(* PLC project ia_tools test project, CODESYS CODESYS V3.5 SP16, author Toni Kucic *)
(* stored: creationDateTime 2021-03-31T21:46:16.9462712, version 1.0, modificationDateTime 2021-03-31T21:46:13.3815902, organization ia_tools *)
(* This is a test project to test and display the ia_tools features *)

TYPE typeDUT1 : STRUCT
  dummy1 : BOOL := TRUE;  (* Dummy variable1 *)
  dummy2 : REAL;  (* Dummy variable2 *)
  dummy3 : typeDUT2;  (* Dummy variable3 *)
  dummy4 : ARRAY[0..2] OF BOOL;  (* Dummy variable4 *)
END_STRUCT;
END_TYPE

TYPE typeDUT2 : STRUCT
  dummy1 : BOOL := TRUE;  (* Dummy variable1 *)
  dummy2 : REAL;  (* Dummy variable2 *)
  dummy3 : typeDUT1;  (* Dummy variable3 *)
  dummy4 : ARRAY[0..2] OF BOOL;  (* Dummy variable4 *)
END_STRUCT;
END_TYPE

(* values of enumTest: member1: Documentation of member 1; member2: Documentation of member 2; member3: Documentation of member 3; member4: Documentation of member 4 without value *)

{attribute 'qualified_only'}
{attribute 'strict'}
TYPE enumTest : (member1 := 0, member2 := 1, member3 := 3, member4);
END_TYPE

TYPE dummyDUT1 : STRUCT
  dummy1 : BOOL := TRUE;  (* Dummy variable1 *)
  dummy2 : REAL;  (* Dummy variable2 *)
  dummy3 : dummyDUT2;  (* Dummy variable3 *)
  dummy4 : ARRAY[0..2] OF BOOL;  (* Dummy variable4 *)
END_STRUCT;
END_TYPE

TYPE dummyDUT2 : STRUCT
  dummy1 : BOOL := TRUE;  (* Dummy variable1 *)
  dummy2 : REAL;  (* Dummy variable2 *)
  dummy3 : dummyDUT1;  (* Dummy variable3 *)
  dummy4 : ARRAY[0..2] OF BOOL;  (* Dummy variable4 *)
END_STRUCT;
END_TYPE

TYPE dummyDUT1 : STRUCT
  dummy1 : BOOL := TRUE;  (* Dummy variable1 *)
  dummy2 : REAL;  (* Dummy variable2 *)
  dummy3 : dummyDUT2;  (* Dummy variable3 *)
  dummy4 : ARRAY[0..2] OF BOOL;  (* Dummy variable4 *)
END_STRUCT;
END_TYPE

TYPE dummyDUT2 : STRUCT
  dummy1 : BOOL := TRUE;  (* Dummy variable1 *)
  dummy2 : REAL;  (* Dummy variable2 *)
  dummy3 : dummyDUT1;  (* Dummy variable3 *)
  dummy4 : ARRAY[0..2] OF BOOL;  (* Dummy variable4 *)
END_STRUCT;
END_TYPE

TYPE DUT : STRUCT

END_STRUCT;
END_TYPE

TYPE dummyDUT1 : STRUCT
  dummy1 : BOOL := TRUE;  (* Dummy variable1 *)
  dummy2 : REAL;  (* Dummy variable2 *)
  dummy3 : dummyDUT2;  (* Dummy variable3 *)
  dummy4 : ARRAY[0..2] OF BOOL;  (* Dummy variable4 *)
END_STRUCT;
END_TYPE

TYPE dummyDUT2 : STRUCT
  dummy1 : BOOL := TRUE;  (* Dummy variable1 *)
  dummy2 : REAL;  (* Dummy variable2 *)
  dummy3 : dummyDUT1;  (* Dummy variable3 *)
  dummy4 : ARRAY[0..2] OF BOOL;  (* Dummy variable4 *)
END_STRUCT;
END_TYPE

TYPE dummyDUT1 : STRUCT
  dummy1 : BOOL := TRUE;  (* Dummy variable1 *)
  dummy2 : REAL;  (* Dummy variable2 *)
  dummy3 : dummyDUT2;  (* Dummy variable3 *)
  dummy4 : ARRAY[0..2] OF BOOL;  (* Dummy variable4 *)
END_STRUCT;
END_TYPE

TYPE dummyDUT2 : STRUCT
  dummy1 : BOOL := TRUE;  (* Dummy variable1 *)
  dummy2 : REAL;  (* Dummy variable2 *)
  dummy3 : dummyDUT1;  (* Dummy variable3 *)
  dummy4 : ARRAY[0..2] OF BOOL;  (* Dummy variable4 *)
END_STRUCT;
END_TYPE

{attribute 'qualified_only'}
VAR_GLOBAL  (* typeGlobalList1 *)
  dummy1 : BOOL := TRUE;  (* Dummy variable1 *)
  dummy2 : REAL;  (* Dummy variable2 *)
  dummy3 : typeDUT1;  (* Dummy variable3 *)
  dummy4 : typeDUT2;  (* Dummy variable4 *)
  dummy5 : ARRAY[0..2] OF BOOL;  (* Dummy variable5 *)
  dummy6 : ARRAY[0..2] OF BOOL := [TRUE, FALSE, TRUE];  (* 1D array with initialization *)
  dummy7 : ARRAY[0..2, 0..3] OF INT;  (* 2D array without initialization *)
  dummy8 : ARRAY[0..2, 0..3] OF INT := [0, 1, 2, 3, 4, 5, 6, 7, 8];  (* 2D array with initialization *)
END_VAR

{attribute 'qualified_only'}
VAR_GLOBAL  (* typeGlobalList2 *)
  dummy1 : BOOL := TRUE;  (* Dummy variable1 *)
  dummy2 : REAL;  (* Dummy variable2 *)
  dummy3 : typeDUT1;  (* Dummy variable3 *)
  dummy4 : typeDUT2;  (* Dummy variable4 *)
  dummy5 : ARRAY[0..2] OF BOOL;  (* Dummy variable5 *)
END_VAR

PROGRAM typeProgram
  VAR_INPUT
    inputVar1 : BOOL;  (* Comment of inputVar1 *)
    inputVar2 : BOOL;  (* Comment of inputVar2 *)
    inputVar3 : POINTER TO BOOL;  (* Comment of inputVar3 as a pointer *)
  END_VAR
  VAR_IN_OUT
    inoutVar1 : BOOL;  (* Comment of inoutVar1 *)
    inoutVar2 : BOOL;  (* Comment of inoutVar2 *)
    inoutVar3 : POINTER TO BOOL;  (* Comment of inoutVar3 as a pointer *)
  END_VAR
  VAR_OUTPUT
    outputVar1 : BOOL;  (* Comment of outputVar1 *)
    outputVar2 : BOOL;  (* Comment of outputVar2 *)
    outputVar3 : POINTER TO BOOL;  (* Comment of outputVar3 as a pointer *)
  END_VAR
  VAR
    localVar1 : BOOL;  (* Comment of localVar1 *)
    localVar2 : BOOL;  (* Comment of localVar2 *)
    localVar3 : POINTER TO BOOL;  (* Local var as a pointer *)
  END_VAR

            (* THIS IS HOW THE CODE LOOKS *)

(*** DOCS STRING EXAMPLE ONE LINE***)
(*** DOCS STRING EXAMPLE
	MULTI
			LINE
			***)
(*** DOCS STRING WITH EMBEDDED CODE *)
outputVar1 := outputVar2;
(* THE CODE ABOVE IS INCLUDED IN THE DOCS ***)

          
END_PROGRAM

FUNCTION_BLOCK typeFunctionBlock
  VAR_INPUT
    inputVar1 : BOOL;  (* Comment of inputVar1 *)
    inputVar2 : BOOL;  (* Comment of inputVar2 *)
    inputVar3 : POINTER TO BOOL;  (* Comment of inputVar3 as a pointer *)
  END_VAR
  VAR_IN_OUT
    inoutVar1 : BOOL;  (* Comment of inoutVar1 *)
    inoutVar2 : BOOL;  (* Comment of inoutVar2 *)
    inoutVar3 : POINTER TO BOOL;  (* Comment of inoutVar3 as a pointer *)
  END_VAR
  VAR_OUTPUT
    outputVar1 : BOOL;  (* Comment of outputVar1 *)
    outputVar2 : BOOL;  (* Comment of outputVar2 *)
    outputVar3 : POINTER TO BOOL;  (* Comment of outputVar3 as a pointer *)
  END_VAR
  VAR
    localVar1 : BOOL;  (* Comment of localVar1 *)
    localVar2 : BOOL;  (* Comment of localVar2 *)
    localVar3 : POINTER TO BOOL;  (* Local var as a pointer *)
  END_VAR

            (* THIS IS HOW THE CODE LOOKS *)

(*** DOCS STRING EXAMPLE ONE LINE***)
(*** DOCS STRING EXAMPLE
	MULTI
			LINE
			***)
(*** DOCS STRING WITH EMBEDDED CODE *)
outputVar1 := outputVar2;
(* THE CODE ABOVE IS INCLUDED IN THE DOCS ***)

          
END_FUNCTION_BLOCK

FUNCTION typeFunction : BOOL
  VAR_INPUT
    inputVar1 : BOOL;  (* Comment of inputVar1 *)
    inputVar2 : BOOL;  (* Comment of inputVar2 *)
    inputVar3 : POINTER TO BOOL;  (* Comment of inputVar3 as a pointer *)
  END_VAR
  VAR_IN_OUT
    inoutVar1 : BOOL;  (* Comment of inoutVar1 *)
    inoutVar2 : BOOL;  (* Comment of inoutVar2 *)
    inoutVar3 : POINTER TO BOOL;  (* Comment of inoutVar3 as a pointer *)
  END_VAR
  VAR_OUTPUT
    outputVar1 : BOOL;  (* Comment of outputVar1 *)
    outputVar2 : BOOL;  (* Comment of outputVar2 *)
    outputVar3 : POINTER TO BOOL;  (* Comment of outputVar3 as a pointer *)
  END_VAR
  VAR
    localVar1 : BOOL;  (* Comment of localVar1 *)
    localVar2 : BOOL;  (* Comment of localVar2 *)
    localVar3 : POINTER TO BOOL;  (* Local var as a pointer to elementary value *)
    localVar4 : POINTER TO enumTest;  (* Local var as a pointer to enumeration *)
    localVar5 : POINTER TO typeDUT1;  (* Local var as a pointer to structure *)
    localVar6 : POINTER TO ARRAY[0..2] OF INT;  (* Local var as a pointer to structure *)
    localVar7 : typeDUT1 := (dummy1 := TRUE, dummy2 := 14.5);  (* Local var, structure with complex init *)
    dummy5 : ARRAY[0..2] OF BOOL;  (* Dummy variable5 *)
    dummy6 : ARRAY[0..2] OF BOOL := [TRUE, FALSE, TRUE];  (* 1D array with initialization *)
    dummy7 : ARRAY[0..2, 0..3] OF INT;  (* 2D array without initialization *)
    dummy8 : ARRAY[0..2, 0..3] OF INT := [0, 1, 2, 3, 4, 5, 6, 7, 8];  (* 2D array with initialization *)
    dummy9 : enumTest;  (* Local variable as enumeration *)
    dummy10 : ARRAY[0..2] OF typeDUT1;  (* Array of user data type *)
    dummy11 : ARRAY[0..2, 0..3, 0..1] OF INT;  (* 3D array without initialization *)
    dummy12 : ARRAY[0..2, 0..3, 0..1] OF INT := [0, 1, 2, 3, 4, 5, 6, 7, 8];  (* 3D array with initialization *)
  END_VAR

            (* THIS IS HOW THE CODE LOOKS *)

(*** DOCS STRING EXAMPLE ONE LINE***)
(*** DOCS STRING EXAMPLE
	MULTI
			LINE
			***)
(*** DOCS STRING WITH EMBEDDED CODE *)
outputVar1 := outputVar2;
(* THE CODE ABOVE IS INCLUDED IN THE DOCS ***)

RETURN;
          
END_FUNCTION

PROGRAM TestProgram_ST
  VAR_INPUT
    inputVar1 : BOOL;  (* Comment of inputVar1 *)
    inputVar2 : BOOL;  (* Comment of inputVar2 *)
    inputVar3 : POINTER TO BOOL;  (* Comment of inputVar3 as a pointer *)
  END_VAR
  VAR_IN_OUT
    inoutVar1 : BOOL;  (* Comment of inoutVar1 *)
    inoutVar2 : BOOL;  (* Comment of inoutVar2 *)
    inoutVar3 : POINTER TO BOOL;  (* Comment of inoutVar3 as a pointer *)
  END_VAR
  VAR_OUTPUT
    outputVar1 : BOOL;  (* Comment of outputVar1 *)
    outputVar2 : BOOL;  (* Comment of outputVar2 *)
    outputVar3 : POINTER TO BOOL;  (* Comment of outputVar3 as a pointer *)
  END_VAR
  VAR
    localVar1 : BOOL;  (* Comment of localVar1 *)
    localVar2 : BOOL;  (* Comment of localVar2 *)
    localVar3 : POINTER TO BOOL;  (* Local var as a pointer *)
  END_VAR

                    (* THIS IS HOW THE CODE LOOKS *)

(*** DOCS STRING EXAMPLE ONE LINE***)
(*** DOCS STRING EXAMPLE
	MULTI
			LINE
			***)
(*** DOCS STRING WITH EMBEDDED CODE *)
outputVar1 := outputVar2;
(* THE CODE ABOVE IS INCLUDED IN THE DOCS ***)

                  
END_PROGRAM

FUNCTION_BLOCK Test_FunctionBlock_ST
  VAR_INPUT
    inputVar1 : BOOL;  (* Comment of inputVar1 *)
    inputVar2 : BOOL;  (* Comment of inputVar2 *)
    inputVar3 : POINTER TO BOOL;  (* Comment of inputVar3 as a pointer *)
  END_VAR
  VAR_IN_OUT
    inoutVar1 : BOOL;  (* Comment of inoutVar1 *)
    inoutVar2 : BOOL;  (* Comment of inoutVar2 *)
    inoutVar3 : POINTER TO BOOL;  (* Comment of inoutVar3 as a pointer *)
  END_VAR
  VAR_OUTPUT
    outputVar1 : BOOL;  (* Comment of outputVar1 *)
    outputVar2 : BOOL;  (* Comment of outputVar2 *)
    outputVar3 : POINTER TO BOOL;  (* Comment of outputVar3 as a pointer *)
  END_VAR
  VAR
    localVar1 : BOOL;  (* Comment of localVar1 *)
    localVar2 : BOOL;  (* Comment of localVar2 *)
    localVar3 : POINTER TO BOOL;  (* Local var as a pointer *)
  END_VAR

                    (* THIS IS HOW THE CODE LOOKS *)

(*** DOCS STRING EXAMPLE ONE LINE***)
(*** DOCS STRING EXAMPLE
	MULTI
			LINE
			***)
(*** DOCS STRING WITH EMBEDDED CODE *)
outputVar1 := outputVar2;
(* THE CODE ABOVE IS INCLUDED IN THE DOCS ***)

                  
END_FUNCTION_BLOCK

FUNCTION TestFunction_ST : BOOL
  VAR_INPUT
    inputVar1 : BOOL;  (* Comment of inputVar1 *)
    inputVar2 : BOOL;  (* Comment of inputVar2 *)
    inputVar3 : POINTER TO BOOL;  (* Comment of inputVar3 as a pointer *)
  END_VAR
  VAR_IN_OUT
    inoutVar1 : BOOL;  (* Comment of inoutVar1 *)
    inoutVar2 : BOOL;  (* Comment of inoutVar2 *)
    inoutVar3 : POINTER TO BOOL;  (* Comment of inoutVar3 as a pointer *)
  END_VAR
  VAR_OUTPUT
    outputVar1 : BOOL;  (* Comment of outputVar1 *)
    outputVar2 : BOOL;  (* Comment of outputVar2 *)
    outputVar3 : POINTER TO BOOL;  (* Comment of outputVar3 as a pointer *)
  END_VAR
  VAR
    localVar1 : BOOL;  (* Comment of localVar1 *)
    localVar2 : BOOL;  (* Comment of localVar2 *)
    localVar3 : POINTER TO BOOL;  (* Local var as a pointer *)
  END_VAR

                    (* THIS IS HOW THE CODE LOOKS *)

(*** DOCS STRING EXAMPLE ONE LINE***)
(*** DOCS STRING EXAMPLE
	MULTI
			LINE
			***)
(*** DOCS STRING WITH EMBEDDED CODE *)
outputVar1 := outputVar2;
(* THE CODE ABOVE IS INCLUDED IN THE DOCS ***)

RETURN;
                  
END_FUNCTION

PROGRAM TestProgram_ST
  VAR_INPUT
    inputVar1 : BOOL;  (* Comment of inputVar1 *)
    inputVar2 : BOOL;  (* Comment of inputVar2 *)
    inputVar3 : POINTER TO BOOL;  (* Comment of inputVar3 as a pointer *)
  END_VAR
  VAR_IN_OUT
    inoutVar1 : BOOL;  (* Comment of inoutVar1 *)
    inoutVar2 : BOOL;  (* Comment of inoutVar2 *)
    inoutVar3 : POINTER TO BOOL;  (* Comment of inoutVar3 as a pointer *)
  END_VAR
  VAR_OUTPUT
    outputVar1 : BOOL;  (* Comment of outputVar1 *)
    outputVar2 : BOOL;  (* Comment of outputVar2 *)
    outputVar3 : POINTER TO BOOL;  (* Comment of outputVar3 as a pointer *)
  END_VAR
  VAR
    localVar1 : BOOL;  (* Comment of localVar1 *)
    localVar2 : BOOL;  (* Comment of localVar2 *)
    localVar3 : POINTER TO BOOL;  (* Local var as a pointer *)
  END_VAR

                    (* THIS IS HOW THE CODE LOOKS *)

(*** DOCS STRING EXAMPLE ONE LINE***)
(*** DOCS STRING EXAMPLE
	MULTI
			LINE
			***)
(*** DOCS STRING WITH EMBEDDED CODE *)
outputVar1 := outputVar2;
(* THE CODE ABOVE IS INCLUDED IN THE DOCS ***)

                  
END_PROGRAM

FUNCTION_BLOCK Test_FunctionBlock_ST
  VAR_INPUT
    inputVar1 : BOOL;  (* Comment of inputVar1 *)
    inputVar2 : BOOL;  (* Comment of inputVar2 *)
    inputVar3 : POINTER TO BOOL;  (* Comment of inputVar3 as a pointer *)
  END_VAR
  VAR_IN_OUT
    inoutVar1 : BOOL;  (* Comment of inoutVar1 *)
    inoutVar2 : BOOL;  (* Comment of inoutVar2 *)
    inoutVar3 : POINTER TO BOOL;  (* Comment of inoutVar3 as a pointer *)
  END_VAR
  VAR_OUTPUT
    outputVar1 : BOOL;  (* Comment of outputVar1 *)
    outputVar2 : BOOL;  (* Comment of outputVar2 *)
    outputVar3 : POINTER TO BOOL;  (* Comment of outputVar3 as a pointer *)
  END_VAR
  VAR
    localVar1 : BOOL;  (* Comment of localVar1 *)
    localVar2 : BOOL;  (* Comment of localVar2 *)
    localVar3 : POINTER TO BOOL;  (* Local var as a pointer *)
  END_VAR

                    (* THIS IS HOW THE CODE LOOKS *)

(*** DOCS STRING EXAMPLE ONE LINE***)
(*** DOCS STRING EXAMPLE
	MULTI
			LINE
			***)
(*** DOCS STRING WITH EMBEDDED CODE *)
outputVar1 := outputVar2;
(* THE CODE ABOVE IS INCLUDED IN THE DOCS ***)

                  
END_FUNCTION_BLOCK

FUNCTION TestFunction_ST : BOOL
  VAR_INPUT
    inputVar1 : BOOL;  (* Comment of inputVar1 *)
    inputVar2 : BOOL;  (* Comment of inputVar2 *)
    inputVar3 : POINTER TO BOOL;  (* Comment of inputVar3 as a pointer *)
  END_VAR
  VAR_IN_OUT
    inoutVar1 : BOOL;  (* Comment of inoutVar1 *)
    inoutVar2 : BOOL;  (* Comment of inoutVar2 *)
    inoutVar3 : POINTER TO BOOL;  (* Comment of inoutVar3 as a pointer *)
  END_VAR
  VAR_OUTPUT
    outputVar1 : BOOL;  (* Comment of outputVar1 *)
    outputVar2 : BOOL;  (* Comment of outputVar2 *)
    outputVar3 : POINTER TO BOOL;  (* Comment of outputVar3 as a pointer *)
  END_VAR
  VAR
    localVar1 : BOOL;  (* Comment of localVar1 *)
    localVar2 : BOOL;  (* Comment of localVar2 *)
    localVar3 : POINTER TO BOOL;  (* Local var as a pointer *)
  END_VAR

                    (* THIS IS HOW THE CODE LOOKS *)

(*** DOCS STRING EXAMPLE ONE LINE***)
(*** DOCS STRING EXAMPLE
	MULTI
			LINE
			***)
(*** DOCS STRING WITH EMBEDDED CODE *)
outputVar1 := outputVar2;
(* THE CODE ABOVE IS INCLUDED IN THE DOCS ***)

RETURN;
                  
END_FUNCTION

FUNCTION TestFunction_ST : BOOL
  VAR_INPUT
    inputVar1 : BOOL;  (* Comment of inputVar1 *)
    inputVar2 : BOOL;  (* Comment of inputVar2 *)
    inputVar3 : POINTER TO BOOL;  (* Comment of inputVar3 as a pointer *)
  END_VAR
  VAR_IN_OUT
    inoutVar1 : BOOL;  (* Comment of inoutVar1 *)
    inoutVar2 : BOOL;  (* Comment of inoutVar2 *)
    inoutVar3 : POINTER TO BOOL;  (* Comment of inoutVar3 as a pointer *)
  END_VAR
  VAR_OUTPUT
    outputVar1 : BOOL;  (* Comment of outputVar1 *)
    outputVar2 : BOOL;  (* Comment of outputVar2 *)
    outputVar3 : POINTER TO BOOL;  (* Comment of outputVar3 as a pointer *)
  END_VAR
  VAR
    localVar1 : BOOL;  (* Comment of localVar1 *)
    localVar2 : BOOL;  (* Comment of localVar2 *)
    localVar3 : POINTER TO BOOL;  (* Local var as a pointer *)
  END_VAR

                    (* THIS IS HOW THE CODE LOOKS *)

(*** DOCS STRING EXAMPLE ONE LINE***)
(*** DOCS STRING EXAMPLE
	MULTI
			LINE
			***)
(*** DOCS STRING WITH EMBEDDED CODE *)
outputVar1 := outputVar2;
(* THE CODE ABOVE IS INCLUDED IN THE DOCS ***)

RETURN;
                  
END_FUNCTION

PROGRAM TestProgram_ST
  VAR_INPUT
    inputVar1 : BOOL;  (* Comment of inputVar1 *)
    inputVar2 : BOOL;  (* Comment of inputVar2 *)
    inputVar3 : POINTER TO BOOL;  (* Comment of inputVar3 as a pointer *)
  END_VAR
  VAR_IN_OUT
    inoutVar1 : BOOL;  (* Comment of inoutVar1 *)
    inoutVar2 : BOOL;  (* Comment of inoutVar2 *)
    inoutVar3 : POINTER TO BOOL;  (* Comment of inoutVar3 as a pointer *)
  END_VAR
  VAR_OUTPUT
    outputVar1 : BOOL;  (* Comment of outputVar1 *)
    outputVar2 : BOOL;  (* Comment of outputVar2 *)
    outputVar3 : POINTER TO BOOL;  (* Comment of outputVar3 as a pointer *)
  END_VAR
  VAR
    localVar1 : BOOL;  (* Comment of localVar1 *)
    localVar2 : BOOL;  (* Comment of localVar2 *)
    localVar3 : POINTER TO BOOL;  (* Local var as a pointer *)
  END_VAR

                    (* THIS IS HOW THE CODE LOOKS *)

(*** DOCS STRING EXAMPLE ONE LINE***)
(*** DOCS STRING EXAMPLE
	MULTI
			LINE
			***)
(*** DOCS STRING WITH EMBEDDED CODE *)
outputVar1 := outputVar2;
(* THE CODE ABOVE IS INCLUDED IN THE DOCS ***)

                  
END_PROGRAM

FUNCTION_BLOCK Test_FunctionBlock_ST
  VAR_INPUT
    inputVar1 : BOOL;  (* Comment of inputVar1 *)
    inputVar2 : BOOL;  (* Comment of inputVar2 *)
    inputVar3 : POINTER TO BOOL;  (* Comment of inputVar3 as a pointer *)
  END_VAR
  VAR_IN_OUT
    inoutVar1 : BOOL;  (* Comment of inoutVar1 *)
    inoutVar2 : BOOL;  (* Comment of inoutVar2 *)
    inoutVar3 : POINTER TO BOOL;  (* Comment of inoutVar3 as a pointer *)
  END_VAR
  VAR_OUTPUT
    outputVar1 : BOOL;  (* Comment of outputVar1 *)
    outputVar2 : BOOL;  (* Comment of outputVar2 *)
    outputVar3 : POINTER TO BOOL;  (* Comment of outputVar3 as a pointer *)
  END_VAR
  VAR
    localVar1 : BOOL;  (* Comment of localVar1 *)
    localVar2 : BOOL;  (* Comment of localVar2 *)
    localVar3 : POINTER TO BOOL;  (* Local var as a pointer *)
  END_VAR

                    (* THIS IS HOW THE CODE LOOKS *)

(*** DOCS STRING EXAMPLE ONE LINE***)
(*** DOCS STRING EXAMPLE
	MULTI
			LINE
			***)
(*** DOCS STRING WITH EMBEDDED CODE *)
outputVar1 := outputVar2;
(* THE CODE ABOVE IS INCLUDED IN THE DOCS ***)

                  
END_FUNCTION_BLOCK

FUNCTION TestFunction_ST : BOOL
  VAR_INPUT
    inputVar1 : BOOL;  (* Comment of inputVar1 *)
    inputVar2 : BOOL;  (* Comment of inputVar2 *)
    inputVar3 : POINTER TO BOOL;  (* Comment of inputVar3 as a pointer *)
  END_VAR
  VAR_IN_OUT
    inoutVar1 : BOOL;  (* Comment of inoutVar1 *)
    inoutVar2 : BOOL;  (* Comment of inoutVar2 *)
    inoutVar3 : POINTER TO BOOL;  (* Comment of inoutVar3 as a pointer *)
  END_VAR
  VAR_OUTPUT
    outputVar1 : BOOL;  (* Comment of outputVar1 *)
    outputVar2 : BOOL;  (* Comment of outputVar2 *)
    outputVar3 : POINTER TO BOOL;  (* Comment of outputVar3 as a pointer *)
  END_VAR
  VAR
    localVar1 : BOOL;  (* Comment of localVar1 *)
    localVar2 : BOOL;  (* Comment of localVar2 *)
    localVar3 : POINTER TO BOOL;  (* Local var as a pointer *)
  END_VAR

                    (* THIS IS HOW THE CODE LOOKS *)

(*** DOCS STRING EXAMPLE ONE LINE***)
(*** DOCS STRING EXAMPLE
	MULTI
			LINE
			***)
(*** DOCS STRING WITH EMBEDDED CODE *)
outputVar1 := outputVar2;
(* THE CODE ABOVE IS INCLUDED IN THE DOCS ***)

RETURN;
                  
END_FUNCTION

PROGRAM TestProgram_ST
  VAR_INPUT
    inputVar1 : BOOL;  (* Comment of inputVar1 *)
    inputVar2 : BOOL;  (* Comment of inputVar2 *)
    inputVar3 : POINTER TO BOOL;  (* Comment of inputVar3 as a pointer *)
  END_VAR
  VAR_IN_OUT
    inoutVar1 : BOOL;  (* Comment of inoutVar1 *)
    inoutVar2 : BOOL;  (* Comment of inoutVar2 *)
    inoutVar3 : POINTER TO BOOL;  (* Comment of inoutVar3 as a pointer *)
  END_VAR
  VAR_OUTPUT
    outputVar1 : BOOL;  (* Comment of outputVar1 *)
    outputVar2 : BOOL;  (* Comment of outputVar2 *)
    outputVar3 : POINTER TO BOOL;  (* Comment of outputVar3 as a pointer *)
  END_VAR
  VAR
    localVar1 : BOOL;  (* Comment of localVar1 *)
    localVar2 : BOOL;  (* Comment of localVar2 *)
    localVar3 : POINTER TO BOOL;  (* Local var as a pointer *)
  END_VAR

                    (* THIS IS HOW THE CODE LOOKS *)

(*** DOCS STRING EXAMPLE ONE LINE***)
(*** DOCS STRING EXAMPLE
	MULTI
			LINE
			***)
(*** DOCS STRING WITH EMBEDDED CODE *)
outputVar1 := outputVar2;
(* THE CODE ABOVE IS INCLUDED IN THE DOCS ***)

                  
END_PROGRAM

FUNCTION_BLOCK Test_FunctionBlock_ST
  VAR_INPUT
    inputVar1 : BOOL;  (* Comment of inputVar1 *)
    inputVar2 : BOOL;  (* Comment of inputVar2 *)
    inputVar3 : POINTER TO BOOL;  (* Comment of inputVar3 as a pointer *)
  END_VAR
  VAR_IN_OUT
    inoutVar1 : BOOL;  (* Comment of inoutVar1 *)
    inoutVar2 : BOOL;  (* Comment of inoutVar2 *)
    inoutVar3 : POINTER TO BOOL;  (* Comment of inoutVar3 as a pointer *)
  END_VAR
  VAR_OUTPUT
    outputVar1 : BOOL;  (* Comment of outputVar1 *)
    outputVar2 : BOOL;  (* Comment of outputVar2 *)
    outputVar3 : POINTER TO BOOL;  (* Comment of outputVar3 as a pointer *)
  END_VAR
  VAR
    localVar1 : BOOL;  (* Comment of localVar1 *)
    localVar2 : BOOL;  (* Comment of localVar2 *)
    localVar3 : POINTER TO BOOL;  (* Local var as a pointer *)
  END_VAR

                    (* THIS IS HOW THE CODE LOOKS *)

(*** DOCS STRING EXAMPLE ONE LINE***)
(*** DOCS STRING EXAMPLE
	MULTI
			LINE
			***)
(*** DOCS STRING WITH EMBEDDED CODE *)
outputVar1 := outputVar2;
(* THE CODE ABOVE IS INCLUDED IN THE DOCS ***)

                  
END_FUNCTION_BLOCK

CONFIGURATION PLC1
  RESOURCE Application1 ON PLC
    {attribute 'qualified_only'}
    VAR_GLOBAL  (* GlobalVars1 *)
      dummy1 : BOOL := TRUE;  (* Dummy variable1 *)
      dummy2 : REAL;  (* Dummy variable2 *)
      dummy3 : dummyDUT1;  (* Dummy variable3 *)
      dummy4 : dummyDUT2;  (* Dummy variable4 *)
      dummy5 : ARRAY[0..2] OF BOOL;  (* Dummy variable5 *)
    END_VAR
    {attribute 'qualified_only'}
    VAR_GLOBAL  (* GlobalVars2 *)
      dummy1 : BOOL := TRUE;  (* Dummy variable1 *)
      dummy2 : REAL;  (* Dummy variable2 *)
      dummy3 : dummyDUT1;  (* Dummy variable3 *)
      dummy4 : dummyDUT2;  (* Dummy variable4 *)
      dummy5 : ARRAY[0..2] OF BOOL;  (* Dummy variable5 *)
    END_VAR
  END_RESOURCE
END_CONFIGURATION

CONFIGURATION PLC2
  RESOURCE Application2 ON PLC
    {attribute 'qualified_only'}
    VAR_GLOBAL  (* GlobalVars1 *)
      dummy1 : BOOL := TRUE;  (* Dummy variable1 *)
      dummy2 : REAL;  (* Dummy variable2 *)
      dummy3 : dummyDUT1;  (* Dummy variable3 *)
      dummy4 : dummyDUT2;  (* Dummy variable4 *)
      dummy5 : ARRAY[0..2] OF BOOL;  (* Dummy variable5 *)
    END_VAR
    {attribute 'qualified_only'}
    VAR_GLOBAL  (* GlobalVars2 *)
      dummy1 : BOOL := TRUE;  (* Dummy variable1 *)
      dummy2 : REAL;  (* Dummy variable2 *)
      dummy3 : dummyDUT1;  (* Dummy variable3 *)
      dummy4 : dummyDUT2;  (* Dummy variable4 *)
      dummy5 : ARRAY[0..2] OF BOOL;  (* Dummy variable5 *)
    END_VAR
  END_RESOURCE
  RESOURCE App ON PLC
    {attribute 'qualified_only'}
    VAR_GLOBAL  (* GlobalVars1 *)
      dummy1 : BOOL := TRUE;  (* Dummy variable1 *)
      dummy2 : REAL;  (* Dummy variable2 *)
      dummy3 : dummyDUT1;  (* Dummy variable3 *)
      dummy4 : dummyDUT2;  (* Dummy variable4 *)
      dummy5 : ARRAY[0..2] OF BOOL;  (* Dummy variable5 *)
    END_VAR
    {attribute 'qualified_only'}
    VAR_GLOBAL  (* GlobalVars2 *)
      dummy1 : BOOL := TRUE;  (* Dummy variable1 *)
      dummy2 : REAL;  (* Dummy variable2 *)
      dummy3 : dummyDUT1;  (* Dummy variable3 *)
      dummy4 : dummyDUT2;  (* Dummy variable4 *)
      dummy5 : ARRAY[0..2] OF BOOL;  (* Dummy variable5 *)
    END_VAR
  END_RESOURCE
  RESOURCE App_1 ON PLC
    {attribute 'qualified_only'}
    VAR_GLOBAL  (* GlobalVars1 *)
      dummy1 : BOOL := TRUE;  (* Dummy variable1 *)
      dummy2 : REAL;  (* Dummy variable2 *)
      dummy3 : dummyDUT1;  (* Dummy variable3 *)
      dummy4 : dummyDUT2;  (* Dummy variable4 *)
      dummy5 : ARRAY[0..2] OF BOOL;  (* Dummy variable5 *)
    END_VAR
    {attribute 'qualified_only'}
    VAR_GLOBAL  (* GlobalVars2 *)
      dummy1 : BOOL := TRUE;  (* Dummy variable1 *)
      dummy2 : REAL;  (* Dummy variable2 *)
      dummy3 : dummyDUT1;  (* Dummy variable3 *)
      dummy4 : dummyDUT2;  (* Dummy variable4 *)
      dummy5 : ARRAY[0..2] OF BOOL;  (* Dummy variable5 *)
    END_VAR
  END_RESOURCE
END_CONFIGURATION
